FUNCTION_BLOCK INTERNAL FB_AdsErrorHelper_Tests EXTENDS FB_TestSuite
VAR_INPUT
END_VAR
VAR_OUTPUT
END_VAR
VAR
END_VAR

Test01_ErrorId10Provided_Expect_ERR_NOIO();
Test02_GetErrorInfo_ERR_NOIO_ExpectCorrectInfo();

METHOD PRIVATE Test01_ErrorId10Provided_Expect_ERR_NOIO
VAR
	eExpectedErrorCode : E_AdsErrorCode := E_AdsErrorCode.ERR_NOIO;
END_VAR
TcUnit.TEST('Test01_ErrorId10Provided_Expect_ERR_NOIO');

AssertEquals_UDINT(
	Actual := AdsErrorHelper.ErrorIdToEnum(10),
	Expected := eExpectedErrorCode,
	Message := 'Conversion from udint to E_AdsErrorCode was incorrect!');

TcUnit.TEST_FINISHED();
END_METHOD

METHOD PRIVATE Test02_GetErrorInfo_ERR_NOIO_ExpectCorrectInfo
VAR_INPUT
END_VAR
TcUnit.TEST('Test02_GetErrorInfo_ERR_NOIO_ExpectCorrectInfo');

AssertEquals_STRING(
	Actual := AdsErrorHelper.GetErrorInfo(eAdsErrorCode := E_AdsErrorCode.ERR_NOIO),
	Expected := 'No IO.',
	Message := 'Error message for the provided error code was not correct!');

TcUnit.TEST_FINISHED();
END_METHOD

END_FUNCTION_BLOCK

(* stored: Version 1.1.0.1, ProductVersion 3.1.4024.13
   POU FB_AdsErrorHelper_Tests: Id {82ab6e93-8e0a-0bec-3ac8-85f5fd4bb181}, SpecialFunc None
   Method Test01_ErrorId10Provided_Expect_ERR_NOIO: Id {66812773-4d6f-02f1-2eec-e1f4bf4667a8}
   Method Test02_GetErrorInfo_ERR_NOIO_ExpectCorrectInfo: Id {2570b377-4117-043d-2aa5-932b4192b491} *)
